// TwinCAT 3 PLC project KoffieZetten
// ProgramVersion: 3.1.4024.0
// libraries:
//   Tc2_Standard, * (Beckhoff Automation GmbH)
//   Tc2_System, * (Beckhoff Automation GmbH)
//   Tc3_Module, * (Beckhoff Automation GmbH)
//   VisuSymbols,3.5.10.0,System
// project tree:
//   / GlobalTextList.TcGTLO, GVL.TcGVL, PlcTask.TcTTO, Visualization Manager.TcVMO (not stored)
//   POUs/ KoffieZetten.TcPOU, MAIN.TcPOU, resetVars.TcPOU
//   VISUs/ Visualization.TcVIS
// real-time tasks:
//   TASK PlcTask: cycle T#10ms, priority 20, ADS port 350

CONFIGURATION KoffieZetten
    RESOURCE PLC ON TwinCAT3
        TASK PlcTask(INTERVAL := T#10ms, PRIORITY := 20);
        PROGRAM MAIN WITH PlcTask : MAIN;
    END_RESOURCE
END_CONFIGURATION

// ---- GVL.TcGVL
VAR_GLOBAL
	//inputs
	filterPlaatsen : BOOL := FALSE;				//De gebruiker plaatst een filter
	waterreservoirVullen : BOOL := FALSE;		//De gebruiker voegt een eenheid water toe, er kunnen meerdere eenheden water toegevoegd worden aan het reservoir
	scoopieDrBij : BOOL := FALSE;				//De gebruiker voegt een schepje filtermaling toe, er kunnen meerdere schepjes toegevoegd worden (variabele is vernoemd naar de bekende uitspraak van Joel Beukers)
	apparaatAanzetten : BOOL := FALSE;			//Het apparaat wordt ingeschakeld/gestart
	ikBenMoe : BOOL := FALSE;					//De staat van zijn van de gebruiker wordt vastgelegd, dit is van belang voor hoe de koffie moet smaken
	allesLegen : BOOL := FALSE;					//De kan wordt geleegd, het filter eruit, alle variabelen worden gereset
		
	//outputs
	apparaatAan : BOOL := FALSE;				//Staat het apparaat aan of niet
	filterGeplaatst : BOOL := FALSE;			//Is er een filter in het apparaat geplaatst?
	aantalSchepjes : INT := 0;					//Houdt bij hoeveel schepjes filtermaling de gebruiker toevoegt
	storeSchepjes: INT;							//Nodig voor het slechts toevoegen van 1 schepje
	reservoirLevel : INT := 0;					//Houdt bij hoeveel water de gebruiker toevoegt
	storeReservoir : INT;						//Nodig voor het slechts toevoegen van 1 level
	koffieKlaar : BOOL := FALSE;				//Koffie is klaar!
	apparaatLeeg : BOOL := TRUE;				//Alle variabelen zijn gereset
	koffieError : BOOL := FALSE;				//Er is een probleem opgetreden
	waterigeKoffie : BOOL := FALSE;				//De koffie is waterig van smaak
	sterkeKoffie : BOOL := FALSE;				//De koffie is sterk van smaak
	lekkereKoffie : BOOL := FALSE;				//De koffie is perfect gelukt!
	state : INT := 1;							//Houdt de staat van het apparaat bij, 1 = uit en 2 = aan
END_VAR

// ---- POUs/MAIN.TcPOU
PROGRAM MAIN
VAR
	
END_VAR


IF GVL.apparaatLeeg THEN
	GVL.state := 1;
	GVL.allesLegen := FALSE;
	GVL.apparaatLeeg := FALSE;
END_IF

CASE state OF
	1: 				//Apparaat staat uit, de gebruiker kan het apparaat vullen
		IF GVL.allesLegen OR (GVL.filterGeplaatst = FALSE AND GVL.aantalSchepjes > 0) THEN
			GVL.koffieError := TRUE;
		END_IF
		
		IF GVL.filterPlaatsen AND NOT GVL.filterGeplaatst THEN
			GVL.filterGeplaatst := TRUE;
		END_IF
		
		IF GVL.scoopieDrBij THEN
			GVL.aantalSchepjes := GVL.storeSchepjes + 1;
			IF GVL.aantalSchepjes > 12 THEN
				GVL.koffieError := TRUE;
			END_IF
		ELSE
			GVL.storeSchepjes := GVL.aantalschepjes;
		END_IF
		
		IF GVL.waterreservoirVullen THEN
			GVL.reservoirLevel := GVL.storeReservoir + 1;
			IF GVL.reservoirLevel > 6 THEN
				GVL.koffieError := TRUE;
			END_IF
		ELSE
			GVL.storeReservoir := GVL.reservoirLevel;
		END_IF
		
		IF GVL.allesLegen THEN
			resetVars();
		END_IF
		
		IF GVL.apparaatAanzetten THEN
			GVL.state := 2;
		END_IF
		
	2: 				//Apparaat staat aan, koffie wordt gezet op basis van de gebruikersinputs
		koffieZetten();
		
END_CASE;

END_PROGRAM

// ---- POUs/resetVars.TcPOU
PROGRAM resetVars
VAR
END_VAR

//inputs
			GVL.filterPlaatsen := FALSE;
			GVL.waterreservoirVullen := FALSE;
			GVL.scoopieDrBij := FALSE;
			GVL.apparaatAanzetten := FALSE;
			GVL.ikBenMoe := FALSE;
			GVL.allesLegen := FALSE;
				
			//outputs
			GVL.apparaatAan := FALSE;
			GVL.filterGeplaatst := FALSE;
			GVL.aantalSchepjes := 0;
			GVL.reservoirLevel := 0;
			GVL.koffieKlaar := FALSE;
			GVL.apparaatLeeg := TRUE;
			GVL.koffieError := FALSE;
			GVL.waterigeKoffie := FALSE;
			GVL.sterkeKoffie := FALSE;
			GVL.lekkereKoffie := FALSE;

END_PROGRAM

// ---- POUs/KoffieZetten.TcPOU
PROGRAM KoffieZetten
VAR
END_VAR

IF GVL.aantalSchepjes = 2*GVL.reservoirLevel THEN
		GVL.lekkereKoffie := TRUE;
	ELSIF GVL.aantalSchepjes < 2*GVL.reservoirLevel THEN
		GVL.waterigeKoffie := TRUE;
	ELSIF GVL.aantalSchepjes > 2*GVL.reservoirLevel THEN
		GVL.sterkeKoffie := TRUE;
	
	IF GVL.ikBenMoe THEN
		GVL.lekkereKoffie := TRUE;
	END_IF
			
END_IF
	GVL.apparaatLeeg := FALSE;
	GVL.koffieKlaar := TRUE;
	
	IF GVL.allesLegen THEN
		resetVars();
	END_IF

END_PROGRAM

// ---- GlobalTextList.TcGTLO
TEXTLIST GlobalTextList
  854 = 'aantalSchepjes'
  424 = 'allesLegen'
  114 = 'Apparaat feedback'
  914 = 'apparaatAan'
  627 = 'apparaatAanzetten'
  567 = 'Apparaatbediening'
  858 = 'apparaatLeeg'
  515 = 'apparaatStarten'
  154 = 'filterGeplaatst'
  672 = 'filterPlaatsen'
  881 = 'Gebruikersinputs'
  380 = 'ikBenMoe'
  420 = 'koffieError'
  444 = 'koffieKlaar'
  130 = 'lekkereKoffie'
  331 = 'reservoirLevel'
  884 = 'Resultaat'
  245 = 'ScoopieDrBij'
  219 = 'sterkeKoffie'
  564 = 'User inputs'
  383 = 'waterigeKoffie'
  736 = 'waterreservoirVullen'
END_TEXTLIST

// ---- VISUs/Visualization.TcVIS
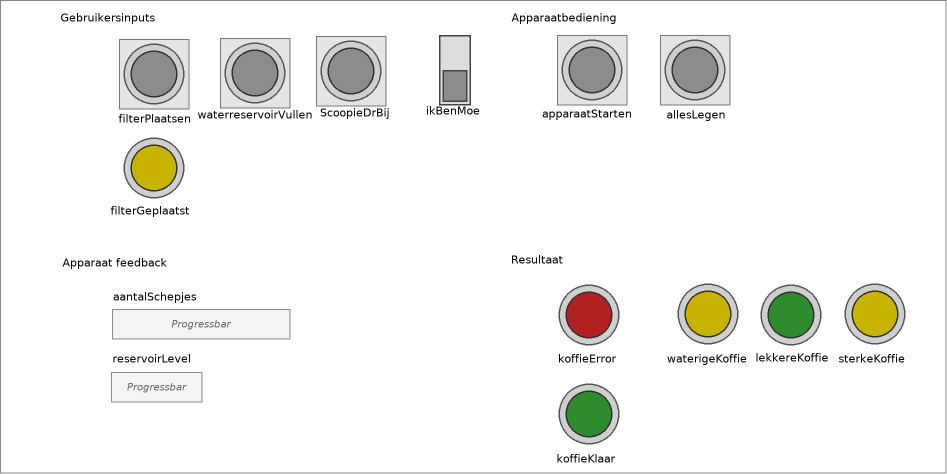
VISUALIZATION Visualization  // 947x474
    Lamp1 (119,133 70x70), variable: MAIN.filterGeplaatst, style: Lamp-Lamp1-Yellow
    Lamp1 (554,379 70x70), variable: MAIN.koffieKlaar, style: Lamp-Lamp1-Green
    Lamp1 (554,280 70x70), variable: MAIN.koffieError, style: Lamp-Lamp1-Red
    Label (512,99 150x30), "apparaatStarten"
    Label (511,444 150x30), "koffieKlaar"
    Label (512,344 150x30), "koffieError"
    Label (75,196 150x30), "filterGeplaatst"
    Label (80,104 150x30), "filterPlaatsen"
    Label (180,100 150x30), "waterreservoirVullen"
    Label (280,98 150x30), "ScoopieDrBij"
    Label (621,100 150x30), "allesLegen"
    DipSwitch (420,35 70x70), variable: MAIN.ikBenMoe, behaviour: TOGGLE, style: Switch-DipSwitch-Gray
    Label (378,96 150x30), "ikBenMoe"
    Lamp1 (756,280 70x70), variable: MAIN.lekkereKoffie, style: Lamp-Lamp1-Green
    Lamp1 (840,279 70x70), variable: MAIN.sterkeKoffie, style: Lamp-Lamp1-Yellow
    Lamp1 (673,279 70x70), variable: MAIN.waterigeKoffie, style: Lamp-Lamp1-Yellow
    Label (797,344 150x30), "sterkeKoffie"
    Label (632,344 150x30), "waterigeKoffie"
    Label (717,343 150x30), "lekkereKoffie"
    Label (80,282 150x30), "aantalSchepjes"
    Label (77,344 150x30), "reservoirLevel"
    PushSwitch (119,39 70x70), variable: GVL.filterPlaatsen, behaviour: TAP, style: Switch-PushSwitch-Gray
    PushSwitch (220,38 70x70), variable: GVL.waterreservoirVullen, behaviour: TAP, style: Switch-PushSwitch-Gray
    PushSwitch (316,36 70x70), variable: GVL.scoopieDrBij, behaviour: TAP, style: Switch-PushSwitch-Gray
    PushSwitch (660,35 70x70), variable: GVL.allesLegen, behaviour: TAP, style: Switch-PushSwitch-Gray
    PushSwitch (557,35 70x70), variable: GVL.apparaatAanzetten, behaviour: TAP, style: Switch-PushSwitch-Gray
    Progressbar (112,309 178x30), variable: aantalSchepjes
    Label (33,3 150x30), "Gebruikersinputs"
    Label (40,248 150x30), "Apparaat feedback"
    Progressbar (111,372 91x30), variable: reservoirLevel
    Label (489,3 150x30), "Apparaatbediening"
    Label (462,245 150x30), "Resultaat"
END_VISUALIZATION
